RoboDK station: wcs_plc_20240624_140000.rdk

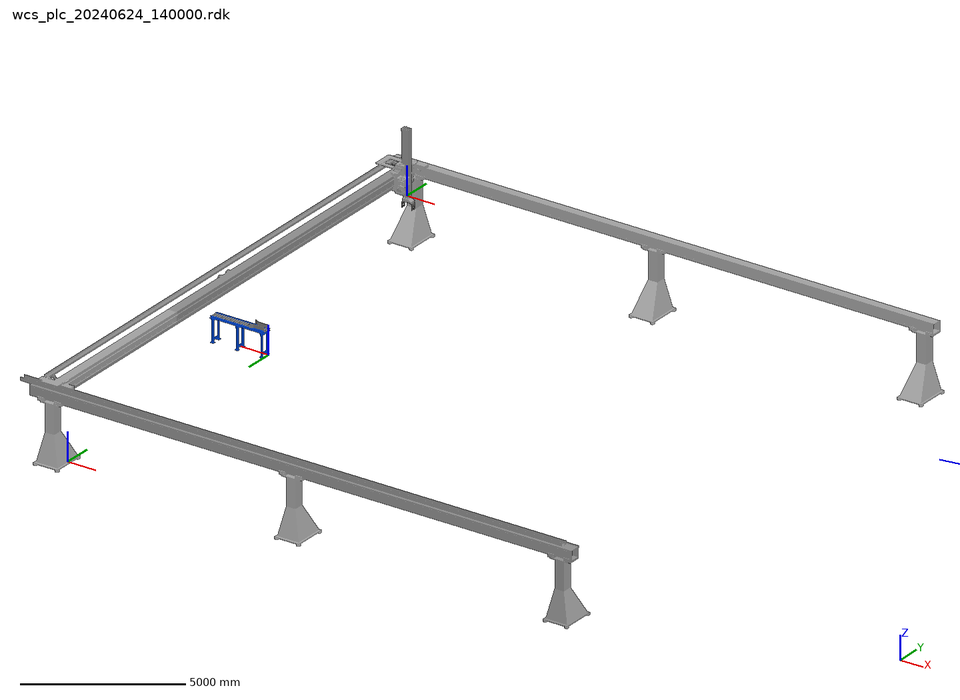
[picture v0: the station drawn from its stored meshes, robots at their saved joint values, targets as dots, program paths as lines]
Station wcs_plc_20240624_140000 (saved by RoboDK 5.6.8). Poses are relative to the parent item; angles as X-Y-Z fixed-axis rotations.
Station parameters (name, value as stored): TAGS, ['Milling']
  - frame conveyor Base at (750, 9500, 0) mm, rotated rx 0 ry 0 rz 180 deg
    - robot conveyor: 1 axes
        modified DH rows (alpha deg, a mm, theta deg, d mm): 0, 0, 0, 0 linear
        base shift (0, 0, 0) mm, rotated rx 0 ry 90 rz 0 deg
        joint limits [-99999] to [9999999]; home [0]; saved at [1000]
      - tool conveyor_TCP, TCP at (160, 110, 135) mm, rotated rx -180 ry 0 rz -180 deg
    - target con_pitch (joint target) at (1000, 0, 880) mm; joints [1000, 0, 0] of conveyor
    - target con_home (joint target) at (160, 110, 1015) mm, rotated rx -180 ry 0 rz -180 deg; joints [0] of conveyor
  - camera Camera 1
  - frame Frame 36 at (25830, 10500, 2900) mm, rotated rx -95 ry 0 rz 90 deg
  - frame gantry Base at (0, 0, 0) mm
    - robot gantry: 3 axes
        modified DH rows (alpha deg, a mm, theta deg, d mm): 0, 0, 0, 0 linear; 90, 0, 90, 0 linear; 90, 0, 0, 0 linear
        base shift (0, 0, 0) mm, rotated rx 0 ry -90 rz 180 deg
        joint limits [-5, -5, -5] to [18000, 17000, 1500]; home [0, 0, 0]; saved at [0, 0, 0]
      - frame gripper Base at (0, 0, 0) mm, rotated rx -180 ry 0 rz 0 deg
        - robot gripper: 1 axes
            modified DH rows (alpha deg, a mm, theta deg, d mm): 0, 0, 0, 0 linear
            base shift (0, 0, 0) mm, rotated rx 0 ry 90 rz 0 deg
            joint limits [-200] to [0]; home [0]; saved at [0]
        - target open_gripper (Cartesian target) at (0, 0, 0) mm; joints [0] of gripper
        - target close_gripper (Cartesian target) at (-55, 0, 0) mm; joints [-55] of gripper
    - target gantry_home (Cartesian target) at (-66.33, 17957.34, 1743.56) mm, rotated rx 180 ry 0 rz 0 deg; joints [0, 0, 0] of gantry
    - target UP_pickup (Cartesian target) at (590, 9400, 1743.56) mm, rotated rx 180 ry 0 rz 0 deg; joints [656.33, 8557.342, 0] of gantry
    - target IN_pickup (Cartesian target) at (590, 9400, 1275) mm, rotated rx 180 ry 0 rz 0 deg; joints [656.33, 8557.34, 468.56] of gantry
    - folder pallet
